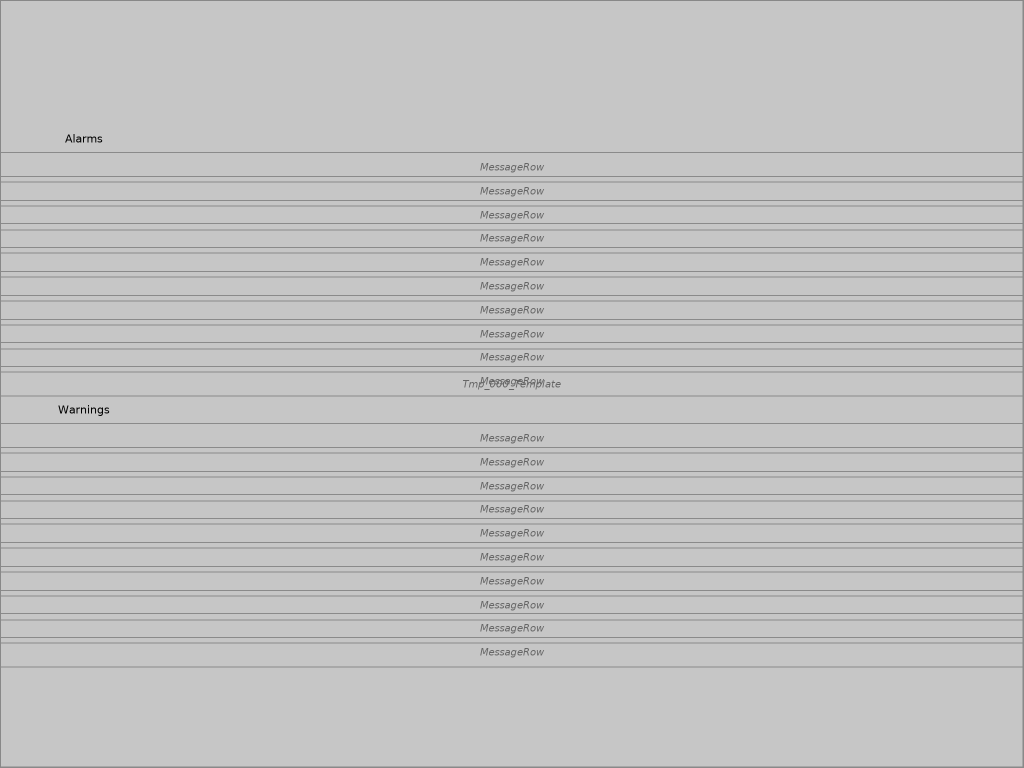
VISUALIZATION Msg_020_Alarms  // 1024x768
    Frame (0,0 1024x768)
        shows Tmp_000_Template(header := gHMIData.hmiHeader)
    Frame (0,152 1024x30)
        shows MessageRow(msg := gHMIData.gAlarmViewMsg.AlarmViewMsg[1])
    Frame (0,176 1024x30)
        shows MessageRow(msg := gHMIData.gAlarmViewMsg.AlarmViewMsg[2])
    Frame (0,200 1024x30)
        shows MessageRow(msg := gHMIData.gAlarmViewMsg.AlarmViewMsg[3])
    Frame (0,223 1024x30)
        shows MessageRow(msg := gHMIData.gAlarmViewMsg.AlarmViewMsg[4])
    Frame (0,247 1024x30)
        shows MessageRow(msg := gHMIData.gAlarmViewMsg.AlarmViewMsg[5])
    Frame (0,271 1024x30)
        shows MessageRow(msg := gHMIData.gAlarmViewMsg.AlarmViewMsg[6])
    Frame (0,295 1024x30)
        shows MessageRow(msg := gHMIData.gAlarmViewMsg.AlarmViewMsg[7])
    Frame (0,319 1024x30)
        shows MessageRow(msg := gHMIData.gAlarmViewMsg.AlarmViewMsg[8])
    Frame (0,342 1024x30)
        shows MessageRow(msg := gHMIData.gAlarmViewMsg.AlarmViewMsg[9])
    Rectangle (9,124 150x30), "Alarms"
    Frame (0,366 1024x30)
        shows MessageRow(msg := gHMIData.gAlarmViewMsg.AlarmViewMsg[10])
    Frame (0,423 1024x30)
        shows MessageRow(msg := gHMIData.gAlarmViewMsg.WarningViewMsg[1])
    Frame (0,447 1024x30)
        shows MessageRow(msg := gHMIData.gAlarmViewMsg.WarningViewMsg[2])
    Frame (0,471 1024x30)
        shows MessageRow(msg := gHMIData.gAlarmViewMsg.WarningViewMsg[3])
    Frame (0,494 1024x30)
        shows MessageRow(msg := gHMIData.gAlarmViewMsg.WarningViewMsg[4])
    Frame (0,518 1024x30)
        shows MessageRow(msg := gHMIData.gAlarmViewMsg.WarningViewMsg[5])
    Frame (0,542 1024x30)
        shows MessageRow(msg := gHMIData.gAlarmViewMsg.WarningViewMsg[6])
    Frame (0,566 1024x30)
        shows MessageRow(msg := gHMIData.gAlarmViewMsg.WarningViewMsg[7])
    Frame (0,590 1024x30)
        shows MessageRow(msg := gHMIData.gAlarmViewMsg.WarningViewMsg[8])
    Frame (0,613 1024x30)
        shows MessageRow(msg := gHMIData.gAlarmViewMsg.WarningViewMsg[9])
    Rectangle (9,395 150x30), "Warnings"
    Frame (0,637 1024x30)
        shows MessageRow(msg := gHMIData.gAlarmViewMsg.WarningViewMsg[10])
END_VISUALIZATION

(* stored: Version 1.1.0.1, ProductVersion 3.1.4024.12
   Visu Msg_020_Alarms: Id {f8834c1c-bbcb-4aa8-8da4-f4c6d4f472f9} *)
